(* IEC 61131-3 sources: plc_projects/SridarRasi/SridarRasi, 6 files *)

(* ---- RasiFoodsGVL.st ---- *)
(* Part 1 of main GVL — HMI / %M tags only. Part 2: scripts/st_v16/GVL_RETAIN_PASTE.st *)
(* Combined: scripts/st_v16/GVL_LIVE_PLANT.st *)
{attribute 'qualified_only'}
VAR_GLOBAL
    Recipe_Weights AT %MD100: ARRAY [1..20] OF REAL;
	Semi_Auto_Bin_Material_Mapping AT %MW60: ARRAY [1..10] OF INT;
	Auto_Bin_Material_Mapping AT %MW50: ARRAY[1..6] OF INT;
	Auto_Coarse_To_Fine_speed AT %MD120: ARRAY[1..6] OF REAL := [1.0,1.0,1.0,1.0,1.0,1.0];
	Auto_Bin_Tolerance AT %MD150: ARRAY[1..6] OF REAL;
	Semi_Auto_Bin_Tolerance AT %MD160: ARRAY[1..10] OF REAL :=[0.2,0.2,0.2,0.2,0.2,0.2,0.2,0.2,0.2,0.2];
	Start_Button AT %MX2.0: BOOL;
	///E_Stop_Active AT %MX2.1: BOOL;
	Next_Cycle_Ready AT %MX2.2: BOOL;
	Reset AT %MX2.3: BOOL;
	Next_Cycle_Start AT %MX2.4: BOOL;
	Auto_Active_Mat AT %MW70: INT;
	Auto_Active_Bin AT %MW71: INT;
	Semi_Auto_Active_Mat AT %MW72: INT;
	Semi_Auto_Active_Bin AT %MW73: INT;
	Target_Batch_Cycles AT %MW74: INT := 0;
	Current_Batch_Cycle AT %MW75: INT;
	Completed_Batch_Cycles AT %MW79: INT;
	Error_Code AT %MW76: INT;
	Run AT %MX2.5 : BOOL;
	load_cell_auto AT %MD174 : REAL;
	load_cell_semi_auto AT %MD175 : REAL;
	Auto_Initial_Tolerance AT %MD176 : REAL := 5.0;
	Semi_Auto_Initial_Tolerance AT %MD178 : REAL := 5.0;
	Empty_Weight_Limit AT %MD186 : REAL := 5.0;
	Ex_Weight_Allow_kg AT %MD188 : REAL := 0.2;
	Auto_Total_Target_Weight AT %MD170 : REAL;
	Semi_Auto_Total_Target_Weight AT %MD171 : REAL;
	Auto_Total_Actual_Weight AT %MD180 : REAL;
	Semi_Auto_Total_Actual_Weight AT %MD184 : REAL;
	Auto_Material_Count AT %MW77: INT;
	Semi_Auto_Material_Count AT %MW78 : INT;
	Auto_Current_Step AT %MW80 : INT;
	Semi_Auto_Current_Step AT %MW81 : INT;
	Auto_Active_Target_Weight AT %MD220 : REAL;
	Semi_Auto_Active_Target_Weight AT %MD224 : REAL;
	Auto_Active_Live_Weight AT %MD172 : REAL;
	Semi_Auto_Active_Live_Weight AT %MD173 : REAL;
	Auto_Excess_Alarm AT %MX2.7 : BOOL;
	Semi_Auto_Excess_Alarm AT %MX2.8 : BOOL;
	Auto_Inter_Bin_Delay AT %MD190 : TIME;
	Semi_Auto_Inter_Bin_Delay AT %MD194 : TIME;
	Auto_Sequence_Complete AT %MX8.2 : BOOL;
	Semi_Auto_Sequence_Complete AT %MX8.3 : BOOL;
	All_Cycles_Complete AT %MX3.2 : BOOL;
	Auto_Status_Message : STRING(80);
	Semi_Auto_Status_Message : STRING(80);
	Auto_Bin : ARRAY[1..6] OF BOOL;
	auto_motor_slow_trigger : ARRAY[1..6] OF BOOL;
	auto_bin_motor : ARRAY[1..6] OF BOOL;
	Semi_Auto_Bin : ARRAY[1..10] OF BOOL;
	Auto_Weights AT %MD300: ARRAY [1..6] OF REAL;
	Semi_Auto_Weights AT %MD350: ARRAY [1..10] OF REAL;
	Auto_Target_Weights AT %MD400: ARRAY [1..6] OF REAL;
	Semi_Auto_Target_Weights AT %MD410: ARRAY [1..10] OF REAL;
	Waiting_Next_batch_HMI_HIDE AT %MX8.1: BOOL;
	All_Cycles_Seq_Completed AT %MX8.4: BOOL;
	Done_Batch_HMI: BOOL;
	Error_bit AT %MX8.5: BOOL;
	Fault_Reset AT %MX8.6: BOOL;
	samyak_weight AT %MD195 : ARRAY[1..4] OF REAL;

END_VAR

(* ---- RasiFoodsPersistant.st ---- *)
VAR_GLOBAL PERSISTENT RETAIN
	(* HMI recipe/mapping shadow — no %M address; restored to GVL after power *)
	Ret_Recipe_Weights: ARRAY [1..20] OF REAL;
	bin_last_weight: REAL;
	Ret_Current_Step: INT;
	Ret_Cycle_Manager_State: INT;
	Ret_Internal_FB_Start: BOOL;
	Ret_bin_last_weight: REAL;
	Ret_GVL_Run: BOOL;
	Ret_Current_Batch_Cycle: INT;
	Ret_Completed_Batch_Cycles: INT;
	Ret_Target_Batch_Cycles: INT;
	Ret_Process_Was_Active: BOOL;
	Ret_Actual_Weights: ARRAY [1..6] OF REAL;
	Ret_Active_Material_ID: INT;
	Ret_Active_Bin_ID: INT;
	Ret_Active_Target_Weight: REAL;
	Ret_Active_Live_Weight: REAL;
	Ret_Resume_Step: INT;
	Ret_Bin_Target_Weights: ARRAY [1..6] OF REAL;
	Ret_Bin_Material_Mapping: ARRAY [1..6] OF INT;
	// Semi-Auto power resume (10 bins; steps 1..10 dosing, 31 settle, 32 complete)
	Ret_Semi_bin_last_weight: REAL;
	Ret_Semi_Current_Step: INT;
	Ret_Semi_Cycle_Manager_State: INT;
	Ret_Semi_Between_Cycle_Hold: BOOL;
	Ret_Semi_Last_Batch_Cycle: INT;
	Ret_Semi_GVL_Run: BOOL;
	Ret_Semi_Current_Batch_Cycle: INT;
	Ret_Semi_Completed_Batch_Cycles: INT;
	Ret_Semi_Target_Batch_Cycles: INT;
	Ret_Semi_Process_Was_Active: BOOL;
	Ret_Semi_Actual_Weights: ARRAY [1..10] OF REAL;
	Ret_Semi_Active_Material_ID: INT;
	Ret_Semi_Active_Bin_ID: INT;
	Ret_Semi_Active_Target_Weight: REAL;
	Ret_Semi_Active_Live_Weight: REAL;
	Ret_Semi_Resume_Step: INT;
	Ret_Semi_Bin_Target_Weights: ARRAY [1..10] OF REAL;
	Ret_Semi_Bin_Material_Mapping: ARRAY [1..10] OF INT;
END_VAR
VAR_GLOBAL PERSISTENT

END_VAR

(* ---- Auto_Batching_V16.st ---- *)
FUNCTION_BLOCK Auto_Batching_V16
VAR_INPUT
    Start_Button : BOOL;                            // Master start command from HMI (%MX2.0)
    Start_PB : BOOL;                                // Physical Start pushbutton DI (one-shot pulse)
    Auto_Mode_DI : BOOL;                            // Auto Mode DI: TRUE = process start allowed; FALSE = HMI/PB start ignored
    E_Stop_Active : BOOL;                           // Emergency Stop circuit status (NC contact: TRUE = Healthy/Run permitted, FALSE = E-Stop tripped)
    Reset : BOOL;                                   // Production abort: clears steps, weights, cycles, CMS.
    Fault_Reset : BOOL;                             // Rising-edge fault acknowledge: clears Error_Code if live fault cleared
    Auto_Bin_Material_Mapping : ARRAY[1..6] OF INT; // Array mapping physical Silos 1..6 to Recipe Material IDs (1..20, 0 = Silo skipped)
    Auto_Coarse_To_Fine_Speed : ARRAY[1..6] OF REAL;// Weight offset threshold (kg) before target to transition from Coarse to Fine feeding
    Auto_Bin_Tolerance : ARRAY[1..6] OF REAL;       // Allowable weight tolerance window (±kg) around target weight for each silo
    Inter_Bin_Delay : TIME := T#5S;                 // Pause after Bin*=FALSE: tailings on SAME bin ID; then next mat (Auto e.g. T#5S)
    Excess_Allowed : BOOL := FALSE;                 // Overfill handling policy: TRUE = proceed if target is exceeded, FALSE = raise alarm and halt
    load_cell_value : REAL;                         // Live gross weight input reading from the Auto scale load cell (kg)
    Target_Batch_Cycles : INT := 1;                 // Target number of batch cycle repetitions configured from HMI (defaults to 1)
    Next_Cycle_Start : BOOL;                        // NextBatchStart: after a completed cycle (Target>1), press when this FB scale < Empty_Weight_Limit
    Empty_Weight_Limit : REAL := 0.5;               // Both scales must be LT this (kg) before Start/Start_PB, Next_Cycle_Start, or Tare pulse
    Line_Fault : BOOL;                              // Auto scale arrLine_Fault. TRUE => Auto_Error_Code=5 + HOLD
    Partner_Line_Fault : BOOL;                      // Partner Semi load-cell comms fail (arrLine_Fault). TRUE => Auto_Error_Code=8
    Partner_Semi_Auto_Bin_Material_Mapping : ARRAY[1..10] OF INT; // Semi silo Mat IDs 1..10 (wire GVL.Semi_Auto_Bin_Material_Mapping)
    Partner_Semi_Sequence_Complete : BOOL;          // Handshake input from Follower (Semi-Auto) Sequence_Complete
END_VAR
VAR_OUTPUT
    Auto_Bin : ARRAY[1..6] OF BOOL;                 // Coarse feeding valve / gate actuation command outputs for Silos 1..6
    auto_motor_slow_trigger : ARRAY[1..6] OF BOOL;  // Fine feeding valve / VFD slow speed command outputs for Silos 1..6
    auto_bin_motor : ARRAY[1..6] OF BOOL;           // Feeder / screw conveyor motor run commands for Silos 1..6
    Actual_Weights : ARRAY[1..6] OF REAL;           // Net material weight (kg) successfully dosed for each silo in the current cycle
    Auto_Sum_Act_Weight : REAL;                     // Sum of Actual_Weights[1..6]
    Auto_Total_Target_Set : ARRAY[1..6] OF REAL;    // Per-bin target kg (bin index 1..6)
    Sequence_Complete : BOOL;                       // Auto Sequence Complete (Step 8 reached)
    Active_Material_ID : INT;                       // Recipe Material ID currently being dosed (1..20, 0 when idle/complete)
    Active_Bin_ID : INT;                            // Physical Silo index currently being dosed (1..6, 0 when idle/complete)
    Active_Target_Weight : REAL;                    // Target weight setpoint (kg) of the ingredient currently being dosed
    Active_Live_Weight : REAL;                      // Live net/tared weight (kg) accumulated into the scale for the active silo
    Current_Step : INT;                             // Real-time sequence step: 0=Idle, 1..6=Dosing, 7=Settle, 8=Complete
    Cycle_Manager_State : INT;                      // Master supervisory state: 0=Idle, 1=Running, 4=All Done, 5=Between Cycles Hold
    Excess_Alarm : BOOL;                            // Overfill alarm

    (* =========================================================================
       MASTER SYSTEM ERROR CODES REFERENCE (Displayed in GVL.Error_Code %MW76):
       0  = System Healthy / No Error
       1  = Auto Duplicate Material ID (within Silos 1..6)
       2  = Auto Invalid Material ID (< 0 or > 20)
       3  = Auto Target Weight < (Coarse_To_Fine_Speed + Tolerance)
       4  = Auto Scale 1 Not Empty (> Empty_Weight_Limit) at Start / Cycle Trigger
       5  = Auto Scale 1 Communication Line Fault (FB_Samyak_Multi Scale 1)
       6  = Recipe / Bin Mapping is all 0s (no ingredients assigned)
       7  = Cross-Scale Duplicate Material (Same Material mapped on Auto and Semi)
       8  = Semi Scale 2 Communication Line Fault (FB_Samyak_Multi Scale 2)
       9  = Semi Duplicate Material ID (within Silos 1..10)
       10 = Semi Scale 2 Not Empty (> Empty_Weight_Limit) at Start / Cycle Trigger
       11 = Semi Invalid Material ID (< 0 or > 20)
       12 = Semi Target Weight < (Coarse_To_Fine_Speed + Tolerance)
       ========================================================================= *)
    Auto_Error_Code : INT;                          // Fault diagnostic code (0=OK, 1..12)
    Error : BOOL;                                   // TRUE when Auto_Error_Code > 0
    Auto_Current_Batch_Cycle : INT;                 // Active batch cycle number currently processing (1..Target_Batch_Cycles)
    Auto_Completed_Batch_Cycles : INT;              // Total number of batch cycle loops completed successfully
    Auto_All_Cycles_Complete : BOOL;                // Master flag: TRUE when all Target_Batch_Cycles have finished
    Partner_Semi_Current_Batch_Cycle : INT;         // Follower (Semi) cycle number mirroring GVL
    Partner_Semi_Completed_Batch_Cycles : INT;      // Follower (Semi) completed cycles
    Partner_Semi_All_Cycles_Complete : BOOL;        // Follower (Semi) all cycles complete flag
    Status_Message : STRING(80);                    // Diagnostic status message
    Tare_Auto_Batch : BOOL;                         // One-scan pulse to Auto scale load cell indicator
    Waiting_Next_Batch : BOOL;                      // TRUE in State 5 between cycles
    Next_Cycle_Ready : BOOL;                        // TRUE when both scales are confirmed empty and debounced in State 5

    // Master-to-Follower Single Coordination Signal
    Master_Run : BOOL;                              // Master Run signal wired directly to Semi-Auto Follower
END_VAR
VAR
    bin_last_weight : REAL;
    actual_bin : REAL;
    target_weight : REAL;
    cutoff_trigger_weight : REAL;
    min_tol_weight : REAL;
    max_tol_weight : REAL;
    Paused_By_Hold : BOOL;
    Effective_Delay : TIME;
    Inter_Bin_Settling : BOOL;
    Inter_Bin_Settle_Arm : INT;
    Inter_Bin_Timer : TON;
    Settle_Hold_Step : INT;
    Settle_Hold_Mat : INT;
    Settle_Hold_Target : REAL;
    Inter_Bin_Next_Step : INT;
    Mat_Idx : INT;
    j_Mat : INT;
    i : INT;
    j : INT;
    Completion_Timer : TON;
    Empty_Debounce_Timer : TON;                     // 1s debounce filter for empty scale verification in State 5
    Internal_FB_Start : BOOL;
    Duplicate_Found : BOOL;
    Duplicate_Vs_Partner : BOOL;
    Duplicate_Partner_Internal : BOOL;
    Auto_Mapping_All_Zero : BOOL;
    Partner_Mapping_All_Zero : BOOL;
    Invalid_Material_Range : BOOL;
    Weight_Limit_Error : BOOL;
    Semi_Invalid_Material_Range : BOOL;
    Semi_Weight_Limit_Error : BOOL;
    eff_empty_limit : REAL;
    Scale_Empty_OK : BOOL;
    Next_Cycle_Last : BOOL;
    Next_Cycle_Rising : BOOL;
    Tare_Pulse_Req : BOOL;
    Start_Cmd : BOOL;
    Start_Cmd_Last : BOOL;
    Start_Pulse : BOOL;
    First_Scan_Done : BOOL;
    Auto_Has_Active_Bins : BOOL;
    Semi_Has_Active_Bins : BOOL;
    Reset_Last : BOOL;
    Reset_Pulse : BOOL;
    Fault_Reset_Last : BOOL;
    Fault_Reset_Pulse : BOOL;
    Between_Cycle_Hold : BOOL;
    Last_Dosing_Step : INT;
    Semi_Sequence_Done : BOOL;
END_VAR

// -----------------------------------------------------------------------------
// 0. TIMINGS, THRESHOLDS & EDGE DETECTION
// -----------------------------------------------------------------------------
Effective_Delay := Inter_Bin_Delay;
IF Effective_Delay = T#0S THEN
    Effective_Delay := T#2S;
END_IF;

eff_empty_limit := Empty_Weight_Limit;
IF eff_empty_limit <= 0.0 THEN
    eff_empty_limit := GVL.Empty_Weight_Limit;
END_IF;
IF eff_empty_limit <= 0.0 THEN
    eff_empty_limit := 0.5;
END_IF;

Scale_Empty_OK := (load_cell_value < eff_empty_limit) AND (GVL.load_cell_auto < eff_empty_limit)
    AND (GVL.load_cell_semi_auto < eff_empty_limit);

Start_Cmd := (Start_Button OR GVL.Start_Button OR Start_PB) AND Auto_Mode_DI;
Start_Pulse := Start_Cmd AND NOT Start_Cmd_Last;
Start_Cmd_Last := Start_Cmd;

Next_Cycle_Rising := (Next_Cycle_Start OR GVL.Next_Cycle_Start) AND NOT Next_Cycle_Last;
Next_Cycle_Last := (Next_Cycle_Start OR GVL.Next_Cycle_Start);

Reset_Pulse := (Reset OR GVL.Reset) AND NOT Reset_Last;
Reset_Last := (Reset OR GVL.Reset);

Fault_Reset_Pulse := Fault_Reset AND NOT Fault_Reset_Last;
Fault_Reset_Last := Fault_Reset;

// Combine direct pin and GVL handshake for Follower completion
Semi_Sequence_Done := Partner_Semi_Sequence_Complete OR GVL.Semi_Auto_Sequence_Complete;

// -----------------------------------------------------------------------------
// 1. FIRST SCAN POWER-RESUME & RETAIN RESTORE
// -----------------------------------------------------------------------------
IF NOT First_Scan_Done THEN
    First_Scan_Done := TRUE;

    // Restore HMI Recipe & Mapping retain if GVL uninitialized
    FOR i := 1 TO 20 DO
        IF (GVL.Recipe_Weights[i] <= 0.001) AND (PersistentVars.Ret_Recipe_Weights[i] > 0.001) THEN
            GVL.Recipe_Weights[i] := PersistentVars.Ret_Recipe_Weights[i];
        END_IF;
    END_FOR;
    FOR i := 1 TO 6 DO
        IF (GVL.Auto_Bin_Material_Mapping[i] = 0) AND (PersistentVars.Ret_Bin_Material_Mapping[i] > 0) THEN
            GVL.Auto_Bin_Material_Mapping[i] := PersistentVars.Ret_Bin_Material_Mapping[i];
        END_IF;
    END_FOR;
    FOR i := 1 TO 10 DO
        IF (GVL.Semi_Auto_Bin_Material_Mapping[i] = 0) AND (PersistentVars.Ret_Semi_Bin_Material_Mapping[i] > 0) THEN
            GVL.Semi_Auto_Bin_Material_Mapping[i] := PersistentVars.Ret_Semi_Bin_Material_Mapping[i];
        END_IF;
    END_FOR;

    // Power Resume: restore exact state without corrupting actual weights with live load cell
    IF PersistentVars.Ret_Process_Was_Active AND (PersistentVars.Ret_Cycle_Manager_State = 1)
       AND (PersistentVars.Ret_Resume_Step >= 1) AND (PersistentVars.Ret_Resume_Step <= 6) THEN

        Current_Step := PersistentVars.Ret_Resume_Step;
        Last_Dosing_Step := Current_Step;
        Cycle_Manager_State := 1;
        Internal_FB_Start := TRUE;
        Between_Cycle_Hold := FALSE;
        GVL.Run := TRUE;
        Master_Run := TRUE;
        GVL.Current_Batch_Cycle := PersistentVars.Ret_Current_Batch_Cycle;
        GVL.Completed_Batch_Cycles := PersistentVars.Ret_Completed_Batch_Cycles;
        IF PersistentVars.Ret_Target_Batch_Cycles > 0 THEN
            GVL.Target_Batch_Cycles := PersistentVars.Ret_Target_Batch_Cycles;
        END_IF;

        bin_last_weight := PersistentVars.Ret_bin_last_weight;
        PersistentVars.bin_last_weight := bin_last_weight;

        // Reconcile with live load cell weight to account for extra material dumped while power was off
        IF (load_cell_value >= bin_last_weight) AND NOT Line_Fault THEN
            Active_Live_Weight := load_cell_value - bin_last_weight;
            Actual_Weights[Current_Step] := Active_Live_Weight;
        ELSE
            Active_Live_Weight := PersistentVars.Ret_Active_Live_Weight;
            Actual_Weights[Current_Step] := Active_Live_Weight;
        END_IF;

        Auto_Sum_Act_Weight := 0.0;
        FOR i := 1 TO 6 DO
            IF i <> Current_Step THEN
                Actual_Weights[i] := PersistentVars.Ret_Actual_Weights[i];
            END_IF;
            GVL.Auto_Weights[i] := Actual_Weights[i];
            Auto_Sum_Act_Weight := Auto_Sum_Act_Weight + Actual_Weights[i];
        END_FOR;
        GVL.Auto_Total_Actual_Weight := Auto_Sum_Act_Weight;

        GVL.Auto_Active_Live_Weight := Active_Live_Weight;
        Active_Material_ID := PersistentVars.Ret_Active_Material_ID;
        Active_Bin_ID := PersistentVars.Ret_Active_Bin_ID;
        Active_Target_Weight := PersistentVars.Ret_Active_Target_Weight;
        GVL.Auto_Active_Mat := Active_Material_ID;
        GVL.Auto_Active_Bin := Active_Bin_ID;
        GVL.Auto_Active_Target_Weight := Active_Target_Weight;

        Paused_By_Hold := TRUE;
        Tare_Pulse_Req := FALSE;
        Tare_Auto_Batch := FALSE;

        // Check if material dumped during power-off has already reached or exceeded target weight
        IF (Active_Target_Weight > 0.0) AND (Active_Live_Weight >= (Active_Target_Weight - Auto_Bin_Tolerance[Current_Step])) THEN
            IF Active_Live_Weight > (Active_Target_Weight + Auto_Bin_Tolerance[Current_Step]) THEN
                Status_Message := CONCAT('Auto [POWER RESUME]: Step ', CONCAT(INT_TO_STRING(Current_Step), ' Overfilled — Waiting Resume'));
            ELSE
                Status_Message := CONCAT('Auto [POWER RESUME]: Step ', CONCAT(INT_TO_STRING(Current_Step), ' Target Reached — Advancing on Resume'));
            END_IF;
        ELSE
            Status_Message := CONCAT('Auto [POWER RESUME]: Step ', CONCAT(INT_TO_STRING(Current_Step), ' Resumed — Ready to Feed'));
        END_IF;

    ELSIF (PersistentVars.Ret_Cycle_Manager_State = 5) THEN
        Cycle_Manager_State := 5;
        Between_Cycle_Hold := TRUE;
        Current_Step := 8;
        Sequence_Complete := TRUE;
        GVL.Auto_Sequence_Complete := TRUE;
        GVL.Run := TRUE;
        Master_Run := TRUE;
        GVL.Current_Batch_Cycle := PersistentVars.Ret_Current_Batch_Cycle;
        GVL.Completed_Batch_Cycles := PersistentVars.Ret_Completed_Batch_Cycles;
        IF PersistentVars.Ret_Target_Batch_Cycles > 0 THEN
            GVL.Target_Batch_Cycles := PersistentVars.Ret_Target_Batch_Cycles;
        END_IF;
        FOR i := 1 TO 6 DO
            Actual_Weights[i] := PersistentVars.Ret_Actual_Weights[i];
            GVL.Auto_Weights[i] := Actual_Weights[i];
        END_FOR;
        Tare_Pulse_Req := FALSE;
        Tare_Auto_Batch := FALSE;
        Status_Message := 'Auto [POWER RESUME]: State 5 - Waiting empty scale & Next_Cycle_Start';

    ELSE
        Current_Step := 0;
        Cycle_Manager_State := 0;
        Internal_FB_Start := FALSE;
        Master_Run := FALSE;
        Between_Cycle_Hold := FALSE;
        Sequence_Complete := FALSE;
        Tare_Pulse_Req := FALSE;
        Tare_Auto_Batch := FALSE;
        Next_Cycle_Ready := FALSE;
        Status_Message := 'Auto [Idle]: Ready - Waiting for Start';
    END_IF;
END_IF;

// Retain snapshot of HMI mappings
FOR i := 1 TO 20 DO
    PersistentVars.Ret_Recipe_Weights[i] := GVL.Recipe_Weights[i];
END_FOR;
FOR i := 1 TO 6 DO
    PersistentVars.Ret_Bin_Material_Mapping[i] := GVL.Auto_Bin_Material_Mapping[i];
END_FOR;
FOR i := 1 TO 10 DO
    PersistentVars.Ret_Semi_Bin_Material_Mapping[i] := GVL.Semi_Auto_Bin_Material_Mapping[i];
END_FOR;

// -----------------------------------------------------------------------------
// 2. CONFIGURATION CHECKS & ERROR DIAGNOSTICS
// -----------------------------------------------------------------------------
Duplicate_Found := FALSE;
Duplicate_Vs_Partner := FALSE;
Duplicate_Partner_Internal := FALSE;
Auto_Mapping_All_Zero := TRUE;
Partner_Mapping_All_Zero := TRUE;
Invalid_Material_Range := FALSE;
Weight_Limit_Error := FALSE;
Auto_Has_Active_Bins := FALSE;
Semi_Has_Active_Bins := FALSE;

GVL.Auto_Total_Target_Weight := 0.0;
GVL.Auto_Material_Count := 0;

FOR i := 1 TO 6 DO
    Mat_Idx := Auto_Bin_Material_Mapping[i];
    IF (Mat_Idx < 1) OR (Mat_Idx > 20) THEN
        Mat_Idx := GVL.Auto_Bin_Material_Mapping[i];
    END_IF;
    IF Mat_Idx <> 0 THEN
        Auto_Mapping_All_Zero := FALSE;
    END_IF;
    IF (Mat_Idx < 0) OR (Mat_Idx > 20) THEN
        Invalid_Material_Range := TRUE;
    END_IF;
    IF (Mat_Idx >= 1) AND (Mat_Idx <= 20) THEN
        FOR j := 1 TO 6 DO
            IF j <> i THEN
                j_Mat := Auto_Bin_Material_Mapping[j];
                IF (j_Mat < 1) OR (j_Mat > 20) THEN
                    j_Mat := GVL.Auto_Bin_Material_Mapping[j];
                END_IF;
                IF (j_Mat = Mat_Idx) THEN
                    Duplicate_Found := TRUE;
                END_IF;
            END_IF;
        END_FOR;
        FOR j := 1 TO 10 DO
            j_Mat := Partner_Semi_Auto_Bin_Material_Mapping[j];
            IF (j_Mat < 1) OR (j_Mat > 20) THEN
                j_Mat := GVL.Semi_Auto_Bin_Material_Mapping[j];
            END_IF;
            IF (j_Mat = Mat_Idx) THEN
                Duplicate_Vs_Partner := TRUE;
            END_IF;
        END_FOR;
        target_weight := GVL.Recipe_Weights[Mat_Idx];
        IF target_weight > 0.0 THEN
            GVL.Auto_Total_Target_Weight := GVL.Auto_Total_Target_Weight + target_weight;
            GVL.Auto_Material_Count := GVL.Auto_Material_Count + 1;
            Auto_Has_Active_Bins := TRUE;
            IF target_weight < (Auto_Coarse_To_Fine_Speed[i] + Auto_Bin_Tolerance[i]) THEN
                Weight_Limit_Error := TRUE;
            END_IF;
        END_IF;
    END_IF;
END_FOR;

Semi_Invalid_Material_Range := FALSE;
Semi_Weight_Limit_Error := FALSE;

FOR i := 1 TO 10 DO
    Mat_Idx := Partner_Semi_Auto_Bin_Material_Mapping[i];
    IF (Mat_Idx < 1) OR (Mat_Idx > 20) THEN
        Mat_Idx := GVL.Semi_Auto_Bin_Material_Mapping[i];
    END_IF;
    IF Mat_Idx <> 0 THEN
        Partner_Mapping_All_Zero := FALSE;
    END_IF;
    IF (Mat_Idx < 0) OR (Mat_Idx > 20) THEN
        Semi_Invalid_Material_Range := TRUE;
    END_IF;
    IF (Mat_Idx >= 1) AND (Mat_Idx <= 20) THEN
        FOR j := 1 TO 10 DO
            IF j <> i THEN
                j_Mat := Partner_Semi_Auto_Bin_Material_Mapping[j];
                IF (j_Mat < 1) OR (j_Mat > 20) THEN
                    j_Mat := GVL.Semi_Auto_Bin_Material_Mapping[j];
                END_IF;
                IF (j_Mat = Mat_Idx) THEN
                    Duplicate_Partner_Internal := TRUE;
                END_IF;
            END_IF;
        END_FOR;
        target_weight := GVL.Recipe_Weights[Mat_Idx];
        IF target_weight > 0.0 THEN
            Semi_Has_Active_Bins := TRUE;
            IF target_weight < GVL.Semi_Auto_Bin_Tolerance[i] THEN
                Semi_Weight_Limit_Error := TRUE;
            END_IF;
        END_IF;
    END_IF;
END_FOR;

IF Line_Fault THEN
    Auto_Error_Code := 5;
    GVL.Error_Code := 5;
    Status_Message := 'Auto_Error_Code 5: Auto Scale 1 Line_Fault Error!';
ELSIF Partner_Line_Fault THEN
    Auto_Error_Code := 8;
    GVL.Error_Code := 8;
    Status_Message := 'Auto_Error_Code 8: Semi Scale 2 Line_Fault Error!';
ELSIF Auto_Mapping_All_Zero AND Partner_Mapping_All_Zero THEN
    Auto_Error_Code := 6;
    GVL.Error_Code := 6;
    Status_Message := 'Auto_Error_Code 6: Mapping is all 0!';
ELSIF Duplicate_Found THEN
    Auto_Error_Code := 1;
    GVL.Error_Code := 1;
    Status_Message := 'Auto_Error_Code 1: Duplicate Material ID within Auto bins!';
ELSIF Duplicate_Partner_Internal THEN
    Auto_Error_Code := 9;
    GVL.Error_Code := 9;
    Status_Message := 'Auto_Error_Code 9: Duplicate Material ID inside Semi mapping!';
ELSIF Duplicate_Vs_Partner THEN
    Auto_Error_Code := 7;
    GVL.Error_Code := 7;
    Status_Message := 'Auto_Error_Code 7: Material ID duplicated on Auto and Semi!';
ELSIF Invalid_Material_Range THEN
    Auto_Error_Code := 2;
    GVL.Error_Code := 2;
    Status_Message := 'Auto_Error_Code 2: Auto Material Index out of range (1..20)!';
ELSIF Semi_Invalid_Material_Range THEN
    Auto_Error_Code := 11;
    GVL.Error_Code := 11;
    Status_Message := 'Auto_Error_Code 11: Semi Material Index out of range (1..20)!';
ELSIF Weight_Limit_Error THEN
    Auto_Error_Code := 3;
    GVL.Error_Code := 3;
    Status_Message := 'Auto_Error_Code 3: Auto Recipe weight < Coarse_To_Fine + Tolerance!';
ELSIF Semi_Weight_Limit_Error THEN
    Auto_Error_Code := 12;
    GVL.Error_Code := 12;
    Status_Message := 'Auto_Error_Code 12: Semi Recipe weight < Tolerance!';
ELSIF (Auto_Error_Code <> 4) AND (Auto_Error_Code <> 10) THEN
    Auto_Error_Code := 0;
    IF (GVL.Error_Code <> 4) AND (GVL.Error_Code <> 10) THEN
        GVL.Error_Code := 0;
    END_IF;
END_IF;

Error := (Auto_Error_Code > 0);

// -----------------------------------------------------------------------------
// 3. MASTER RESET & FAULT RESET
// -----------------------------------------------------------------------------
IF Reset_Pulse THEN
    FOR i := 1 TO 6 DO
        Auto_Bin[i] := FALSE;
        auto_motor_slow_trigger[i] := FALSE;
        auto_bin_motor[i] := FALSE;
        Actual_Weights[i] := 0.0;
        Auto_Total_Target_Set[i] := 0.0;
        GVL.Auto_Bin[i] := FALSE;
        GVL.auto_motor_slow_trigger[i] := FALSE;
        GVL.auto_bin_motor[i] := FALSE;
        GVL.Auto_Weights[i] := 0.0;
        GVL.Auto_Target_Weights[i] := 0.0;
        PersistentVars.Ret_Actual_Weights[i] := 0.0;
        PersistentVars.Ret_Bin_Target_Weights[i] := 0.0;
    END_FOR;
    Auto_Sum_Act_Weight := 0.0;
    GVL.Auto_Total_Actual_Weight := 0.0;
    Sequence_Complete := FALSE;
    GVL.Auto_Sequence_Complete := FALSE;
    Active_Material_ID := 0;
    Active_Bin_ID := 0;
    Active_Target_Weight := 0.0;
    Active_Live_Weight := 0.0;
    GVL.Auto_Active_Target_Weight := 0.0;
    GVL.Auto_Active_Live_Weight := 0.0;
    GVL.Auto_Active_Mat := 0;
    GVL.Auto_Active_Bin := 0;
    Excess_Alarm := FALSE;
    Auto_Error_Code := 0;
    GVL.Error_Code := 0;
    Error := FALSE;
    GVL.Current_Batch_Cycle := 0;
    GVL.Completed_Batch_Cycles := 0;
    GVL.All_Cycles_Complete := FALSE;
    Auto_Completed_Batch_Cycles := 0;
    Auto_Current_Batch_Cycle := 0;
    Auto_All_Cycles_Complete := FALSE;
    GVL.Target_Batch_Cycles := 0;
    GVL.Start_Button := FALSE;
    GVL.Run := FALSE;
    Master_Run := FALSE;
    GVL.Next_Cycle_Start := FALSE;
    Next_Cycle_Ready := FALSE;
    GVL.Next_Cycle_Ready := FALSE;
    Current_Step := 0;
    Cycle_Manager_State := 0;
    Internal_FB_Start := FALSE;
    Tare_Pulse_Req := FALSE;
    Tare_Auto_Batch := FALSE;
    Waiting_Next_Batch := FALSE;
    Between_Cycle_Hold := FALSE;
    Paused_By_Hold := FALSE;
    PersistentVars.Ret_Process_Was_Active := FALSE;
    PersistentVars.Ret_Cycle_Manager_State := 0;
    PersistentVars.Ret_Current_Step := 0;
    PersistentVars.Ret_Resume_Step := 0;
    PersistentVars.Ret_bin_last_weight := 0.0;
    PersistentVars.bin_last_weight := 0.0;
    bin_last_weight := 0.0;
    Status_Message := 'Auto [Reset]: System Reset complete. Ready for Start.';
    RETURN;
END_IF;

IF Fault_Reset_Pulse THEN
    IF (Auto_Error_Code = 4) AND (load_cell_value < eff_empty_limit) AND (GVL.load_cell_auto < eff_empty_limit) THEN
        Auto_Error_Code := 0;
        GVL.Error_Code := 0;
    ELSIF (Auto_Error_Code = 10) AND (GVL.load_cell_semi_auto < eff_empty_limit) THEN
        Auto_Error_Code := 0;
        GVL.Error_Code := 0;
    ELSIF (Auto_Error_Code = 5) AND (NOT Line_Fault) THEN
        Auto_Error_Code := 0;
        GVL.Error_Code := 0;
        Paused_By_Hold := FALSE;
    ELSIF (Auto_Error_Code = 8) AND (NOT Partner_Line_Fault) THEN
        Auto_Error_Code := 0;
        GVL.Error_Code := 0;
        Paused_By_Hold := FALSE;
    END_IF;
    Error := (Auto_Error_Code > 0);
END_IF;

// Process HOLD on Safety / Fault conditions
IF NOT E_Stop_Active OR NOT Auto_Mode_DI OR (Auto_Error_Code > 0) THEN
    Paused_By_Hold := TRUE;
    FOR i := 1 TO 6 DO
        Auto_Bin[i] := FALSE;
        auto_motor_slow_trigger[i] := FALSE;
        auto_bin_motor[i] := FALSE;
        GVL.Auto_Bin[i] := FALSE;
        GVL.auto_motor_slow_trigger[i] := FALSE;
        GVL.auto_bin_motor[i] := FALSE;
    END_FOR;
ELSE
    Paused_By_Hold := FALSE;
END_IF;

// -----------------------------------------------------------------------------
// 4. MASTER CYCLE MANAGER STATE MACHINE
// -----------------------------------------------------------------------------
CASE Cycle_Manager_State OF
    0: // IDLE
        Internal_FB_Start := FALSE;
        Master_Run := FALSE;
        IF NOT PersistentVars.Ret_Process_Was_Active THEN
            GVL.Run := FALSE;
        END_IF;
        GVL.Next_Cycle_Start := FALSE;
        Next_Cycle_Ready := FALSE;
        GVL.Next_Cycle_Ready := FALSE;
        Sequence_Complete := FALSE;
        GVL.Auto_Sequence_Complete := FALSE;
        Current_Step := 0;
        GVL.Auto_Current_Step := 0;

        IF Start_Pulse THEN
            IF Target_Batch_Cycles > 0 THEN
                GVL.Target_Batch_Cycles := Target_Batch_Cycles;
            ELSIF GVL.Target_Batch_Cycles <= 0 THEN
                GVL.Target_Batch_Cycles := 1;
            END_IF;

            IF NOT E_Stop_Active THEN
                Status_Message := 'Auto [State 0]: Cannot Start - E-Stop Open!';
            ELSIF Auto_Error_Code > 0 AND Auto_Error_Code <> 4 AND Auto_Error_Code <> 10 THEN
                Status_Message := CONCAT('Auto [State 0]: Cannot Start - Error ', INT_TO_STRING(Auto_Error_Code));
            ELSIF (load_cell_value >= eff_empty_limit) OR (GVL.load_cell_auto >= eff_empty_limit) THEN
                Auto_Error_Code := 4;
                GVL.Error_Code := 4;
                Status_Message := CONCAT('Auto [State 0]: Error 4 - Auto Scale 1 not empty (< ', CONCAT(REAL_TO_STRING(eff_empty_limit), ' kg)'));
            ELSIF GVL.load_cell_semi_auto >= eff_empty_limit THEN
                Auto_Error_Code := 10;
                GVL.Error_Code := 10;
                Status_Message := CONCAT('Auto [State 0]: Error 10 - Semi Scale 2 not empty (< ', CONCAT(REAL_TO_STRING(eff_empty_limit), ' kg)'));
            ELSE
                Auto_Error_Code := 0;
                GVL.Error_Code := 0;
                GVL.Current_Batch_Cycle := 1;
                GVL.Completed_Batch_Cycles := 0;
                GVL.All_Cycles_Complete := FALSE;
                Auto_Completed_Batch_Cycles := 0;
                Auto_Current_Batch_Cycle := 1;
                Auto_All_Cycles_Complete := FALSE;

                // Continuous Run Active
                GVL.Run := TRUE;
                Master_Run := TRUE;
                Internal_FB_Start := TRUE;
                Cycle_Manager_State := 1;
                Current_Step := 0;

                bin_last_weight := 0.0;
                PersistentVars.bin_last_weight := 0.0;
                PersistentVars.Ret_bin_last_weight := 0.0;
                FOR i := 1 TO 6 DO
                    Actual_Weights[i] := 0.0;
                    PersistentVars.Ret_Actual_Weights[i] := 0.0;
                END_FOR;

                Tare_Pulse_Req := TRUE;
                GVL.Start_Button := FALSE;
            END_IF;
        END_IF;

    1: // RUNNING ACTIVE BATCH CYCLE
        Internal_FB_Start := TRUE;
        GVL.Run := TRUE;
        Master_Run := TRUE;
        GVL.Next_Cycle_Start := FALSE;
        Next_Cycle_Ready := FALSE;
        GVL.Next_Cycle_Ready := FALSE;

        // Dual-Sequence Completion Handshake: BOTH Auto and Semi must finish
        IF Sequence_Complete AND Semi_Sequence_Done AND (Auto_Has_Active_Bins OR Semi_Has_Active_Bins) THEN
            GVL.Completed_Batch_Cycles := GVL.Current_Batch_Cycle;
            Auto_Completed_Batch_Cycles := GVL.Current_Batch_Cycle;

            IF (GVL.Current_Batch_Cycle < GVL.Target_Batch_Cycles) AND (GVL.Error_Code = 0) THEN
                Internal_FB_Start := FALSE;
                Cycle_Manager_State := 5; // Transition to Between-Cycle Hold (Discharge)
                Between_Cycle_Hold := TRUE;
                // GVL.Run remains TRUE continuously throughout State 5
                Status_Message := 'Auto [Cycle Done]: Discharging hoppers - waiting for empty scale';
            ELSE
                Cycle_Manager_State := 4; // All Target Cycles Completed
                Between_Cycle_Hold := FALSE;
                GVL.Start_Button := FALSE;
            END_IF;
        END_IF;

    5: // PAUSED BETWEEN CYCLES (DISCHARGE & NEXT CYCLE READY HANDSHAKE)
        Internal_FB_Start := FALSE;
        GVL.Run := TRUE; // REMAINS TRUE until All_Cycles_Complete
        Master_Run := TRUE;

        // 1-Second Debounce filter for empty scale check
        IF (load_cell_value <= eff_empty_limit) AND (GVL.load_cell_auto <= eff_empty_limit) AND (GVL.load_cell_semi_auto <= eff_empty_limit) THEN
            Empty_Debounce_Timer(IN := TRUE, PT := T#1S);
            IF Empty_Debounce_Timer.Q THEN
                Next_Cycle_Ready := TRUE;
                GVL.Next_Cycle_Ready := TRUE;
                Status_Message := 'Auto [State 5]: Hoppers Empty - Ready for Next Cycle Start';
            END_IF;
        ELSE
            Empty_Debounce_Timer(IN := FALSE);
            Next_Cycle_Ready := FALSE;
            GVL.Next_Cycle_Ready := FALSE;
            Status_Message := CONCAT('Auto [State 5]: Discharging batch (Scale > ', CONCAT(REAL_TO_STRING(eff_empty_limit), ' kg)...'));
        END_IF;

        // Next Cycle Trigger Pulse
        IF Next_Cycle_Rising THEN
            IF Auto_Error_Code > 0 THEN
                Status_Message := CONCAT('Auto [State 5]: Blocked by Auto_Error_Code ', INT_TO_STRING(Auto_Error_Code));
            ELSIF Next_Cycle_Ready AND (GVL.Current_Batch_Cycle < GVL.Target_Batch_Cycles) THEN
                Next_Cycle_Ready := FALSE;
                GVL.Next_Cycle_Ready := FALSE;
                GVL.Next_Cycle_Start := FALSE;
                Next_Cycle_Last := FALSE;

                GVL.Current_Batch_Cycle := GVL.Current_Batch_Cycle + 1;
                Auto_Current_Batch_Cycle := GVL.Current_Batch_Cycle;

                Sequence_Complete := FALSE;
                GVL.Auto_Sequence_Complete := FALSE;
                GVL.Semi_Auto_Sequence_Complete := FALSE;
                Between_Cycle_Hold := FALSE;
                Cycle_Manager_State := 1;
                Current_Step := 0;
                Internal_FB_Start := TRUE;

                bin_last_weight := 0.0;
                PersistentVars.bin_last_weight := 0.0;
                PersistentVars.Ret_bin_last_weight := 0.0;
                FOR i := 1 TO 6 DO
                    Actual_Weights[i] := 0.0;
                    PersistentVars.Ret_Actual_Weights[i] := 0.0;
                    Auto_Bin[i] := FALSE;
                    auto_motor_slow_trigger[i] := FALSE;
                    auto_bin_motor[i] := FALSE;
                END_FOR;

                Tare_Pulse_Req := TRUE;
                Status_Message := CONCAT('Auto [State 5]: Cycle ', CONCAT(INT_TO_STRING(GVL.Current_Batch_Cycle), ' Started'));
            ELSE
                Status_Message := CONCAT('Auto [State 5]: Empty scale < ', CONCAT(REAL_TO_STRING(eff_empty_limit), ' kg before pressing Next Cycle!'));
            END_IF;
        END_IF;

    4: // ALL TARGET BATCH CYCLES COMPLETE
        Internal_FB_Start := FALSE;
        Between_Cycle_Hold := FALSE;
        GVL.Run := FALSE; // Turn off GVL.Run only when all cycles finish
        Master_Run := FALSE;
        GVL.Start_Button := FALSE;
        Auto_All_Cycles_Complete := TRUE;
        GVL.All_Cycles_Complete := TRUE;
        Sequence_Complete := TRUE;
        GVL.Auto_Sequence_Complete := TRUE;
        Next_Cycle_Ready := FALSE;
        GVL.Next_Cycle_Ready := FALSE;
        Status_Message := CONCAT('Auto [Finished]: All ', CONCAT(INT_TO_STRING(GVL.Target_Batch_Cycles), ' Batch Cycles Complete'));

        IF Start_Pulse THEN
            IF Scale_Empty_OK THEN
                Current_Step := 0;
                Cycle_Manager_State := 0;
                Auto_All_Cycles_Complete := FALSE;
                GVL.All_Cycles_Complete := FALSE;
            ELSE
                Auto_Error_Code := 4;
                GVL.Error_Code := 4;
                Status_Message := 'Auto [Finished]: Empty hopper before starting new job!';
            END_IF;
        END_IF;
END_CASE;

// -----------------------------------------------------------------------------
// 5. AUTO DOSING SEQUENCE (STEPS 1..6, SETTLE 7, COMPLETE 8)
// -----------------------------------------------------------------------------
IF (Current_Step = 0) AND Internal_FB_Start AND (Cycle_Manager_State = 1) THEN
    IF NOT Auto_Has_Active_Bins THEN
        Current_Step := 8;
        Sequence_Complete := TRUE;
        GVL.Auto_Sequence_Complete := TRUE;
    ELSE
        Current_Step := 1;
        bin_last_weight := load_cell_value;
        PersistentVars.Ret_bin_last_weight := bin_last_weight;
        PersistentVars.bin_last_weight := bin_last_weight;
        Last_Dosing_Step := 1;
        Sequence_Complete := FALSE;
        GVL.Auto_Sequence_Complete := FALSE;
    END_IF;
END_IF;

CASE Current_Step OF
    0:
        Active_Material_ID := 0;
        Active_Bin_ID := 0;
        Active_Target_Weight := 0.0;
        Active_Live_Weight := 0.0;
        FOR i := 1 TO 6 DO
            Auto_Bin[i] := FALSE;
            auto_motor_slow_trigger[i] := FALSE;
            auto_bin_motor[i] := FALSE;
        END_FOR;

    1..6:
        WHILE (Current_Step >= 1) AND (Current_Step <= 6) DO
            Mat_Idx := Auto_Bin_Material_Mapping[Current_Step];
            IF (Mat_Idx < 1) OR (Mat_Idx > 20) THEN
                Mat_Idx := GVL.Auto_Bin_Material_Mapping[Current_Step];
            END_IF;
            target_weight := 0.0;
            IF (Mat_Idx >= 1) AND (Mat_Idx <= 20) THEN
                target_weight := GVL.Recipe_Weights[Mat_Idx];
            END_IF;

            IF (Mat_Idx < 1) OR (Mat_Idx > 20) OR (target_weight <= 0.0) THEN
                Auto_Bin[Current_Step] := FALSE;
                auto_motor_slow_trigger[Current_Step] := FALSE;
                auto_bin_motor[Current_Step] := FALSE;
                Actual_Weights[Current_Step] := 0.0;
                IF Current_Step = 6 THEN
                    Current_Step := 7;
                    EXIT;
                ELSE
                    Current_Step := Current_Step + 1;
                END_IF;
            ELSE
                EXIT;
            END_IF;
        END_WHILE;

        IF Inter_Bin_Settling THEN
            FOR i := 1 TO 6 DO
                Auto_Bin[i] := FALSE;
                auto_motor_slow_trigger[i] := FALSE;
                auto_bin_motor[i] := FALSE;
            END_FOR;
            Active_Material_ID := Settle_Hold_Mat;
            Active_Bin_ID := Settle_Hold_Step;
            Active_Target_Weight := Settle_Hold_Target;

            // If held on Excess_Alarm and Excess_Allowed is enabled, clear alarm and advance
            IF Excess_Alarm AND Excess_Allowed THEN
                Excess_Alarm := FALSE;
                bin_last_weight := load_cell_value;
                PersistentVars.Ret_bin_last_weight := bin_last_weight;
                PersistentVars.bin_last_weight := bin_last_weight;
                Current_Step := Inter_Bin_Next_Step;
                Last_Dosing_Step := Current_Step;
                Inter_Bin_Settling := FALSE;
                Inter_Bin_Settle_Arm := 0;
            ELSIF NOT Excess_Alarm THEN
                IF Inter_Bin_Settle_Arm = 0 THEN
                    Inter_Bin_Timer(IN := FALSE);
                    Inter_Bin_Settle_Arm := 1;
                ELSE
                    Inter_Bin_Timer(IN := TRUE, PT := Effective_Delay);
                    IF Inter_Bin_Timer.Q THEN
                        Inter_Bin_Timer(IN := FALSE);

                        // Post-settling final weight check (accounts for in-flight tailings / scale stabilization)
                        actual_bin := load_cell_value - bin_last_weight;
                        IF actual_bin < 0.0 THEN
                            actual_bin := 0.0;
                        END_IF;
                        Actual_Weights[Settle_Hold_Step] := actual_bin;
                        Active_Live_Weight := actual_bin;

                        min_tol_weight := Settle_Hold_Target - Auto_Bin_Tolerance[Settle_Hold_Step];
                        max_tol_weight := Settle_Hold_Target + Auto_Bin_Tolerance[Settle_Hold_Step];

                        IF actual_bin > max_tol_weight THEN
                            IF Excess_Allowed THEN
                                Excess_Alarm := FALSE;
                                bin_last_weight := load_cell_value;
                                PersistentVars.Ret_bin_last_weight := bin_last_weight;
                                PersistentVars.bin_last_weight := bin_last_weight;
                                Current_Step := Inter_Bin_Next_Step;
                                Last_Dosing_Step := Current_Step;
                                Inter_Bin_Settling := FALSE;
                                Inter_Bin_Settle_Arm := 0;
                            ELSE
                                Excess_Alarm := TRUE;
                                Status_Message := CONCAT('Auto [Step ', CONCAT(INT_TO_STRING(Settle_Hold_Step), ']: Settled Overfill Alarm!'));
                            END_IF;
                        ELSIF actual_bin < min_tol_weight THEN
                            // If settled weight is below minimum tolerance, resume fine feeding to top up
                            Inter_Bin_Settling := FALSE;
                            Inter_Bin_Settle_Arm := 0;
                            Excess_Alarm := FALSE;
                            Status_Message := CONCAT('Auto [Step ', CONCAT(INT_TO_STRING(Settle_Hold_Step), ']: Settled below Tol — Topping up'));
                        ELSE
                            // Settled within tolerance range: record final weight and advance to next bin
                            Excess_Alarm := FALSE;
                            bin_last_weight := load_cell_value;
                            PersistentVars.Ret_bin_last_weight := bin_last_weight;
                            PersistentVars.bin_last_weight := bin_last_weight;
                            Current_Step := Inter_Bin_Next_Step;
                            Last_Dosing_Step := Current_Step;
                            Inter_Bin_Settling := FALSE;
                            Inter_Bin_Settle_Arm := 0;
                        END_IF;
                    END_IF;
                END_IF;
            END_IF;

        ELSIF (Current_Step >= 1) AND (Current_Step <= 6) THEN
            Mat_Idx := Auto_Bin_Material_Mapping[Current_Step];
            IF (Mat_Idx < 1) OR (Mat_Idx > 20) THEN
                Mat_Idx := GVL.Auto_Bin_Material_Mapping[Current_Step];
            END_IF;
            target_weight := GVL.Recipe_Weights[Mat_Idx];

            IF Current_Step <> Last_Dosing_Step THEN
                bin_last_weight := load_cell_value;
                PersistentVars.Ret_bin_last_weight := bin_last_weight;
                PersistentVars.bin_last_weight := bin_last_weight;
                Last_Dosing_Step := Current_Step;
            END_IF;

            cutoff_trigger_weight := target_weight - Auto_Coarse_To_Fine_Speed[Current_Step];
            min_tol_weight := target_weight - Auto_Bin_Tolerance[Current_Step];
            max_tol_weight := target_weight + Auto_Bin_Tolerance[Current_Step];

            actual_bin := load_cell_value - bin_last_weight;
            IF actual_bin < 0.0 THEN
                actual_bin := 0.0;
            END_IF;

            Active_Material_ID := Mat_Idx;
            Active_Bin_ID := Current_Step;
            Active_Target_Weight := target_weight;

            // Continually track live weight during both Run and Safety Hold (captures extra power-off dump)
            Actual_Weights[Current_Step] := actual_bin;
            Active_Live_Weight := actual_bin;

            IF (NOT Paused_By_Hold) AND GVL.Run AND (Auto_Error_Code = 0) THEN
                IF actual_bin < cutoff_trigger_weight THEN
                    Auto_Bin[Current_Step] := TRUE;
                    auto_motor_slow_trigger[Current_Step] := FALSE;
                    auto_bin_motor[Current_Step] := TRUE;
                    Excess_Alarm := FALSE;
                    Status_Message := CONCAT('Auto [Step ', CONCAT(INT_TO_STRING(Current_Step), ']: Coarse Feeding'));
                ELSIF actual_bin < min_tol_weight THEN
                    Auto_Bin[Current_Step] := FALSE;
                    auto_motor_slow_trigger[Current_Step] := TRUE;
                    auto_bin_motor[Current_Step] := TRUE;
                    Excess_Alarm := FALSE;
                    Status_Message := CONCAT('Auto [Step ', CONCAT(INT_TO_STRING(Current_Step), ']: Fine Feeding'));
                ELSIF actual_bin > max_tol_weight THEN
                    Auto_Bin[Current_Step] := FALSE;
                    auto_motor_slow_trigger[Current_Step] := FALSE;
                    auto_bin_motor[Current_Step] := FALSE;
                    IF Excess_Allowed THEN
                        Excess_Alarm := FALSE;
                        Status_Message := CONCAT('Auto [Step ', CONCAT(INT_TO_STRING(Current_Step), ']: Target Reached (Excess Allowed)'));
                        Settle_Hold_Step := Current_Step;
                        Settle_Hold_Mat := Mat_Idx;
                        Settle_Hold_Target := target_weight;
                        IF Current_Step >= 6 THEN
                            Current_Step := 7;
                        ELSE
                            Inter_Bin_Next_Step := Current_Step + 1;
                            Inter_Bin_Settling := TRUE;
                            Inter_Bin_Settle_Arm := 0;
                        END_IF;
                    ELSE
                        Excess_Alarm := TRUE;
                        Status_Message := CONCAT('Auto [Step ', CONCAT(INT_TO_STRING(Current_Step), ']: Excess Weight Alarm!'));
                    END_IF;
                ELSE
                    Auto_Bin[Current_Step] := FALSE;
                    auto_motor_slow_trigger[Current_Step] := FALSE;
                    auto_bin_motor[Current_Step] := FALSE;
                    Excess_Alarm := FALSE;
                    Status_Message := CONCAT('Auto [Step ', CONCAT(INT_TO_STRING(Current_Step), ']: Target Reached - Advancing'));
                    Settle_Hold_Step := Current_Step;
                    Settle_Hold_Mat := Mat_Idx;
                    Settle_Hold_Target := target_weight;
                    IF Current_Step >= 6 THEN
                        Current_Step := 7;
                    ELSE
                        Inter_Bin_Next_Step := Current_Step + 1;
                        Inter_Bin_Settling := TRUE;
                        Inter_Bin_Settle_Arm := 0;
                    END_IF;
                END_IF;
            END_IF;
        END_IF;

    7: // FINAL SETTLING DELAY
        Active_Material_ID := 0;
        Active_Bin_ID := 0;
        Active_Target_Weight := 0.0;
        Active_Live_Weight := 0.0;
        FOR i := 1 TO 6 DO
            Auto_Bin[i] := FALSE;
            auto_motor_slow_trigger[i] := FALSE;
            auto_bin_motor[i] := FALSE;
        END_FOR;
        Status_Message := 'Auto [Step 7]: Settling Delay in progress...';
        Completion_Timer(IN := TRUE, PT := Effective_Delay);
        IF Completion_Timer.Q THEN
            Completion_Timer(IN := FALSE);
            Current_Step := 8;
        END_IF;

    8: // AUTO SEQUENCE COMPLETE (WAITS FOR FOLLOWER ASYNCHRONOUSLY)
        Active_Material_ID := 0;
        Active_Bin_ID := 0;
        Active_Target_Weight := 0.0;
        Active_Live_Weight := 0.0;
        FOR i := 1 TO 6 DO
            Auto_Bin[i] := FALSE;
            auto_motor_slow_trigger[i] := FALSE;
            auto_bin_motor[i] := FALSE;
        END_FOR;
        Sequence_Complete := TRUE;
        GVL.Auto_Sequence_Complete := TRUE;
        IF NOT Semi_Sequence_Done THEN
            Status_Message := 'Auto [Step 8]: Auto Finished — Waiting for Semi-Auto to complete...';
        ELSE
            Status_Message := 'Auto [Step 8]: Both Sequences Complete';
        END_IF;
END_CASE;

// -----------------------------------------------------------------------------
// 6. OUTPUT SYNCHRONIZATION & PERSISTENT SNAPSHOT
// -----------------------------------------------------------------------------
FOR i := 1 TO 6 DO
    GVL.Auto_Bin[i] := Auto_Bin[i];
    GVL.auto_motor_slow_trigger[i] := auto_motor_slow_trigger[i];
    GVL.auto_bin_motor[i] := auto_bin_motor[i];
    GVL.Auto_Weights[i] := Actual_Weights[i];
END_FOR;

Auto_Sum_Act_Weight := 0.0;
FOR i := 1 TO 6 DO
    Auto_Sum_Act_Weight := Auto_Sum_Act_Weight + Actual_Weights[i];
END_FOR;
GVL.Auto_Total_Actual_Weight := Auto_Sum_Act_Weight;

GVL.Auto_Active_Mat := Active_Material_ID;
GVL.Auto_Active_Bin := Active_Bin_ID;
GVL.Auto_Active_Target_Weight := Active_Target_Weight;
GVL.Auto_Active_Live_Weight := Active_Live_Weight;
GVL.Auto_Current_Step := Current_Step;
GVL.Auto_Excess_Alarm := Excess_Alarm;

FOR i := 1 TO 6 DO
    Mat_Idx := Auto_Bin_Material_Mapping[i];
    IF (Mat_Idx < 1) OR (Mat_Idx > 20) THEN
        Mat_Idx := GVL.Auto_Bin_Material_Mapping[i];
    END_IF;
    target_weight := 0.0;
    IF (Mat_Idx >= 1) AND (Mat_Idx <= 20) THEN
        target_weight := GVL.Recipe_Weights[Mat_Idx];
    END_IF;
    Auto_Total_Target_Set[i] := target_weight;
    GVL.Auto_Target_Weights[i] := target_weight;
END_FOR;

// Persistent Snapshot
IF Cycle_Manager_State = 4 THEN
    PersistentVars.Ret_Process_Was_Active := FALSE;
    PersistentVars.Ret_Cycle_Manager_State := 0;
    PersistentVars.Ret_Current_Step := 0;
    PersistentVars.Ret_Resume_Step := 0;
    PersistentVars.Ret_Active_Live_Weight := 0.0;
    PersistentVars.Ret_bin_last_weight := 0.0;
    FOR i := 1 TO 6 DO
        PersistentVars.Ret_Actual_Weights[i] := 0.0;
    END_FOR;
ELSIF Cycle_Manager_State = 1 OR Cycle_Manager_State = 5 THEN
    PersistentVars.Ret_Process_Was_Active := TRUE;
    PersistentVars.Ret_Cycle_Manager_State := Cycle_Manager_State;
    PersistentVars.Ret_Current_Step := Current_Step;
    IF (Current_Step >= 1) AND (Current_Step <= 6) THEN
        PersistentVars.Ret_Resume_Step := Current_Step;
    END_IF;
    PersistentVars.Ret_Current_Batch_Cycle := GVL.Current_Batch_Cycle;
    PersistentVars.Ret_Completed_Batch_Cycles := GVL.Completed_Batch_Cycles;
    PersistentVars.Ret_Target_Batch_Cycles := GVL.Target_Batch_Cycles;
    PersistentVars.Ret_Active_Material_ID := Active_Material_ID;
    PersistentVars.Ret_Active_Bin_ID := Active_Bin_ID;
    PersistentVars.Ret_Active_Target_Weight := Active_Target_Weight;
    PersistentVars.Ret_Active_Live_Weight := Active_Live_Weight;
    PersistentVars.Ret_bin_last_weight := bin_last_weight;
    FOR i := 1 TO 6 DO
        PersistentVars.Ret_Actual_Weights[i] := Actual_Weights[i];
    END_FOR;
END_IF;

// -----------------------------------------------------------------------------
// 7. TARE PULSE EMISSION (STRICT INTERLOCK)
// -----------------------------------------------------------------------------
IF Tare_Pulse_Req THEN
    IF Scale_Empty_OK AND (Cycle_Manager_State = 1) AND (Current_Step <= 1) THEN
        Tare_Auto_Batch := TRUE;
    ELSE
        Tare_Auto_Batch := FALSE;
    END_IF;
    Tare_Pulse_Req := FALSE;
ELSE
    Tare_Auto_Batch := FALSE;
END_IF;

Waiting_Next_Batch := (Cycle_Manager_State = 5) AND (GVL.Target_Batch_Cycles > 1) AND (GVL.Current_Batch_Cycle < GVL.Target_Batch_Cycles);
GVL.Waiting_Next_batch_HMI_HIDE := Waiting_Next_Batch;
Auto_Current_Batch_Cycle := GVL.Current_Batch_Cycle;
Auto_Completed_Batch_Cycles := GVL.Completed_Batch_Cycles;
Auto_All_Cycles_Complete := GVL.All_Cycles_Complete;
Partner_Semi_Current_Batch_Cycle := GVL.Current_Batch_Cycle;
Partner_Semi_Completed_Batch_Cycles := GVL.Completed_Batch_Cycles;
Partner_Semi_All_Cycles_Complete := GVL.All_Cycles_Complete;
END_FUNCTION_BLOCK
